// TIA Portal V16 program export: 1 tag tables, 0 data types, 0 data blocks, 1 code blocks (in call order from the OBs), 1 instance data blocks

VAR_GLOBAL   // PLC tag table "Counter_Table"
   stop AT %I0.0 : Bool;
   start AT %I0.1 : Bool;
   system AT %M0.0 : Bool;
   box_conveyor AT %Q0.0 : Bool;
   box_sensor AT %I0.2 : Bool;
   apple_conveyor AT %Q0.1 : Bool;
   apple_sensor AT %I0.3 : Bool;
END_VAR

ORGANIZATION_BLOCK "Counter_Project"   // OB1, LAD, ProgramCycle
TITLE = "Main Program Sweep (Cycle)"
{ S7_Optimized_Access := 'TRUE' }
VERSION : 0.1
// stored: AutoNumber true, IsIECCheckEnabled false, SetENOAutomatically false
   VAR_INPUT
      Initial_Call : Bool;   // Initial call of this OB
      Remanence : Bool;   // =True, if remanent data are available
   END_VAR
BEGIN

REGION Network 1
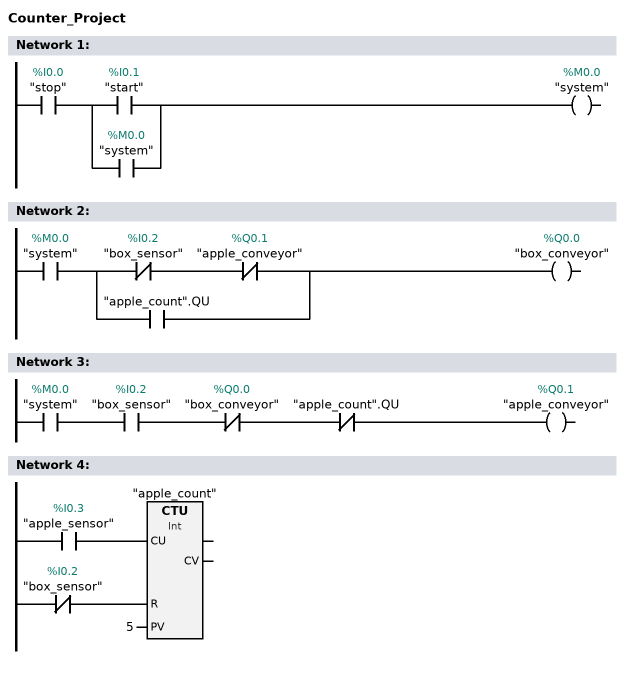
   RUNG wire#powerrail
      Contact( "stop" )
      wire#w1
      Contact( "start" )
      wire#w2
      Coil( "system" )
   END_RUNG
   RUNG wire#w1
      Contact( "system" )
   END_RUNG wire#w2
   // the same network as SCL:
   "system" := "stop" AND ("start" OR "system");
END_REGION

REGION Network 2
   RUNG wire#powerrail
      Contact( "system" )
      wire#w1
      I_Contact( "box_sensor" )
      I_Contact( "apple_conveyor" )
      wire#w2
      Coil( "box_conveyor" )
   END_RUNG
   RUNG wire#w1
      Contact( "apple_count".QU )
   END_RUNG wire#w2
   // the same network as SCL:
   "box_conveyor" := "system" AND ((NOT "box_sensor" AND NOT "apple_conveyor") OR "apple_count".QU);
END_REGION

REGION Network 3
   RUNG wire#powerrail
      Contact( "system" )
      Contact( "box_sensor" )
      I_Contact( "box_conveyor" )
      I_Contact( "apple_count".QU )
      Coil( "apple_conveyor" )
   END_RUNG
   // the same network as SCL:
   "apple_conveyor" := "system" AND "box_sensor" AND NOT "box_conveyor" AND NOT "apple_count".QU;
END_REGION

REGION Network 4
   RUNG wire#powerrail
      Contact( "apple_sensor" )
      { S7_Templates := "value_type := Int" } "apple_count".CTU(r := wire#w1, pv := 5, cv =>)
   END_RUNG
   RUNG wire#powerrail
      I_Contact( "box_sensor" )
   END_RUNG wire#w1
   // the same network as SCL:
   "apple_count".CTU(CU := "apple_sensor", R := NOT "box_sensor", PV := 5);
END_REGION
END_ORGANIZATION_BLOCK

DATA_BLOCK "apple_count"   // DB1
{ S7_Optimized_Access := 'TRUE' }
// stored: AutoNumber true, DBAccessibleFromOPCUA true, InstanceOfName IEC_COUNTER, OfSystemLibElement IEC_COUNTER, OfSystemLibVersion 1.0
"IEC_COUNTER"
   // VAR RETAIN
   //    CU : Bool;
   //    CD : Bool;
   //    R : Bool;
   //    LD : Bool;
   //    QU : Bool;
   //    QD : Bool;
   //    PV : Int;
   //    CV : Int;
   // END_VAR
BEGIN
END_DATA_BLOCK
